FUNCTION F_LogError : STRING;
VAR_INPUT
   Message : T_MaxString;
END_VAR

F_LogError := F_Logger(ADSLOG_MSGTYPE_ERROR, Message);

END_FUNCTION

(* stored: Version 1.1.0.1, ProductVersion 3.1.4026.12
   POU F_LogError: Id {72d2693c-d7be-0c99-2cc7-5909ac95e450}, SpecialFunc None *)
